// TIA Portal V17 export
// export: Created 2024-08-07T21:44:04.708432Z, ExportSetting WithDefaults, DisplayName Totally Integrated Automation Portal, DisplayVersion V17 Update 7, DisplayName TIA Portal Openness, DisplayVersion V17 Update 7, DisplayName TIA Portal Version Control Interface, DisplayVersion V17, DisplayName SINAMICS Startdrive Advanced, DisplayVersion V17 SP2, DisplayName SINAMICS Startdrive G110M, G120, G120C, G120D, G120P, G115D, DisplayVersion V17 SP2, DisplayName SINAMICS Startdrive G130, G150, S120, S150, SINAMICS MV, S210, DisplayVersion V17 SP2, DisplayName STEP 7 Professional, DisplayVersion V17 Update 7, DisplayName STEP 7 Safety, DisplayVersion V17 Update 6, DisplayName WinCC Advanced / Unified PC, DisplayVersion V17 Update 7
DATA_BLOCK "AutoPositions"   // DB11
{ S7_Optimized_Access := 'TRUE' }
VERSION : 0.1
// stored: AutoNumber true, DBAccessibleFromOPCUA true, DBAccessibleFromWebserver true, IsOnlyStoredInLoadMemory false, IsRetainMemResEnabled false, IsWriteProtectedInAS false, MemoryReserve 100
   VAR RETAIN
      St1_Table1 : "UDT_PositionData";
      St2_Table2 : "UDT_PositionData";
      St3_Fitting : "UDT_PositionData";
      R1_Gripper : "UDT_PositionData";
      AE_Gripper : "UDT_PositionData";
      St4_OKposition : "UDT_PositionData";
   END_VAR
   VAR
      emptyPos : "UDT_PositionData";
   END_VAR
BEGIN
   St1_Table1.PartPresent := TRUE;
   St1_Table1.PartNOK := FALSE;
   St1_Table1.PartErrors[0..255] := FALSE;
   St1_Table1.Reference := 0;
   St1_Table1.FinishedOperations[0..15] := FALSE;
   St1_Table1.StFinished[0..15] := FALSE;
   St1_Table1.Scan := '';
   St1_Table1.IJCType := 0;
   St2_Table2.PartPresent := TRUE;
   St2_Table2.PartNOK := FALSE;
   St2_Table2.PartErrors[0..255] := FALSE;
   St2_Table2.Reference := 0;
   St2_Table2.FinishedOperations[0..15] := FALSE;
   St2_Table2.StFinished[0] := FALSE;
   St2_Table2.StFinished[1] := TRUE;
   St2_Table2.StFinished[2..15] := FALSE;
   St2_Table2.Scan := '';
   St2_Table2.IJCType := 0;
   St3_Fitting.PartPresent := FALSE;
   St3_Fitting.PartNOK := FALSE;
   St3_Fitting.PartErrors[0..255] := FALSE;
   St3_Fitting.Reference := 0;
   St3_Fitting.FinishedOperations[0..15] := FALSE;
   St3_Fitting.StFinished[0..15] := FALSE;
   St3_Fitting.Scan := '';
   St3_Fitting.IJCType := 0;
   R1_Gripper.PartPresent := FALSE;
   R1_Gripper.PartNOK := FALSE;
   R1_Gripper.PartErrors[0..255] := FALSE;
   R1_Gripper.Reference := 0;
   R1_Gripper.FinishedOperations[0..15] := FALSE;
   R1_Gripper.StFinished[0..15] := FALSE;
   R1_Gripper.Scan := '';
   R1_Gripper.IJCType := 0;
   AE_Gripper.PartPresent := FALSE;
   AE_Gripper.PartNOK := FALSE;
   AE_Gripper.PartErrors[0..255] := FALSE;
   AE_Gripper.Reference := 0;
   AE_Gripper.FinishedOperations[0..15] := FALSE;
   AE_Gripper.StFinished[0..15] := FALSE;
   AE_Gripper.Scan := '';
   AE_Gripper.IJCType := 0;
   St4_OKposition.PartPresent := TRUE;
   St4_OKposition.PartNOK := FALSE;
   St4_OKposition.PartErrors[0..255] := FALSE;
   St4_OKposition.Reference := 0;
   St4_OKposition.FinishedOperations[0..15] := FALSE;
   St4_OKposition.StFinished[0] := FALSE;
   St4_OKposition.StFinished[1] := TRUE;
   St4_OKposition.StFinished[2] := FALSE;
   St4_OKposition.StFinished[3] := TRUE;
   St4_OKposition.StFinished[4..15] := FALSE;
   St4_OKposition.Scan := '';
   St4_OKposition.IJCType := 0;
   emptyPos.PartPresent := FALSE;
   emptyPos.PartNOK := FALSE;
   emptyPos.PartErrors[0..255] := FALSE;
   emptyPos.Reference := 0;
   emptyPos.FinishedOperations[0..15] := FALSE;
   emptyPos.StFinished[0..15] := FALSE;
   emptyPos.Scan := '';
   emptyPos.IJCType := 0;
END_DATA_BLOCK
